// TIA Portal V19 export
DATA_BLOCK "InfeedPAC3200"   // DB19
TITLE = Instance DB of basic data collection
// Instance DB of basic data collection
// stored: InstanceOfName EnS_EnergyDataBasic, InstanceOfType FB
"EnS_EnergyDataBasic"
   // VAR_INPUT
   //    energyMeta : "EnS_typeEnergyMeta";
   //    energyBasic : "EnS_typeEnergyBasic";
   //    bufferDB { ExternalAccessible := 'False'; ExternalVisible := 'False'; ExternalWritable := 'False'} : DB_ANY;
   //    sD : Variant;
   //    messageSuppress { ExternalAccessible := 'False'; ExternalVisible := 'False'; ExternalWritable := 'False'} : Bool;
   // END_VAR
   // VAR_OUTPUT
   //    error { ExternalAccessible := 'False'; ExternalVisible := 'False'; ExternalWritable := 'False'} : Bool;
   //    errorAlarm1 { ExternalAccessible := 'False'; ExternalVisible := 'False'; ExternalWritable := 'False'} : Bool;
   //    errorAlarm2 { ExternalAccessible := 'False'; ExternalVisible := 'False'; ExternalWritable := 'False'} : Bool;
   //    errorAlarm3 { ExternalAccessible := 'False'; ExternalVisible := 'False'; ExternalWritable := 'False'} : Bool;
   //    alarmState1 { ExternalAccessible := 'False'; ExternalVisible := 'False'; ExternalWritable := 'False'} : Byte;
   //    alarmState2 { ExternalAccessible := 'False'; ExternalVisible := 'False'; ExternalWritable := 'False'} : Byte;
   //    alarmState3 { ExternalAccessible := 'False'; ExternalVisible := 'False'; ExternalWritable := 'False'} : Byte;
   //    status { ExternalAccessible := 'False'; ExternalVisible := 'False'; ExternalWritable := 'False'} : Word;
   //    status1 { ExternalAccessible := 'False'; ExternalVisible := 'False'; ExternalWritable := 'False'} : Word;
   //    status2 { ExternalAccessible := 'False'; ExternalVisible := 'False'; ExternalWritable := 'False'} : Word;
   //    status3 { ExternalAccessible := 'False'; ExternalVisible := 'False'; ExternalWritable := 'False'} : Word;
   //    statusAlarm1 { ExternalAccessible := 'False'; ExternalVisible := 'False'; ExternalWritable := 'False'} : Word;
   //    statusAlarm2 { ExternalAccessible := 'False'; ExternalVisible := 'False'; ExternalWritable := 'False'} : Word;
   //    statusAlarm3 { ExternalAccessible := 'False'; ExternalVisible := 'False'; ExternalWritable := 'False'} : Word;
   // END_VAR
   // VAR_IN_OUT
   //    orgData : "EnS_typeOrgData";
   //    bufferWork : "EnS_typeBufferWork";
   // END_VAR
   // VAR
   //    Program_Alarm1 { ExternalAccessible := 'False'; ExternalVisible := 'False'; ExternalWritable := 'False'; S7_SetPoint := 'True'} : Program_Alarm;
   //    Program_Alarm2 { ExternalAccessible := 'False'; ExternalVisible := 'False'; ExternalWritable := 'False'; S7_SetPoint := 'True'} : Program_Alarm;
   //    Program_Alarm3 { ExternalAccessible := 'False'; ExternalVisible := 'False'; ExternalWritable := 'False'; S7_SetPoint := 'True'} : Program_Alarm;
   //    ss_BufferWrite { ExternalAccessible := 'False'; ExternalVisible := 'False'; ExternalWritable := 'False'; S7_SetPoint := 'True'} : "EnS_BufferWrite";
   //    ss_DataEnergy { ExternalAccessible := 'False'; ExternalVisible := 'False'; ExternalWritable := 'False'; S7_SetPoint := 'True'} : "EnS_typeBufferWriteCtrl";
   //    ss_DataPower { ExternalAccessible := 'False'; ExternalVisible := 'False'; ExternalWritable := 'False'; S7_SetPoint := 'True'} : "EnS_typeBufferWriteCtrl";
   //    ss_DataEnergyCounter { ExternalAccessible := 'False'; ExternalVisible := 'False'; ExternalWritable := 'False'; S7_SetPoint := 'True'} : "EnS_typeBufferWriteCtrl";
   //    si16_CycleWrite { ExternalAccessible := 'False'; ExternalVisible := 'False'; ExternalWritable := 'False'} : Int;
   //    si16_CycleWriteAct { ExternalAccessible := 'False'; ExternalVisible := 'False'; ExternalWritable := 'False'} : Int;
   //    sbo_Write { ExternalAccessible := 'False'; ExternalVisible := 'False'; ExternalWritable := 'False'} : Bool;
   //    sbo_WriteEnergy { ExternalAccessible := 'False'; ExternalVisible := 'False'; ExternalWritable := 'False'} : Bool;
   //    sbo_WritePower { ExternalAccessible := 'False'; ExternalVisible := 'False'; ExternalWritable := 'False'} : Bool;
   //    sbo_WriteEnergyCounter { ExternalAccessible := 'False'; ExternalVisible := 'False'; ExternalWritable := 'False'} : Bool;
   //    sbo_WriteEnergyBusy { ExternalAccessible := 'False'; ExternalVisible := 'False'; ExternalWritable := 'False'} : Bool;
   //    sbo_WritePowerBusy { ExternalAccessible := 'False'; ExternalVisible := 'False'; ExternalWritable := 'False'} : Bool;
   //    sbo_WriteEnergyCounterBusy { ExternalAccessible := 'False'; ExternalVisible := 'False'; ExternalWritable := 'False'} : Bool;
   //    sbo_SyncPulseOld { ExternalAccessible := 'False'; ExternalVisible := 'False'; ExternalWritable := 'False'} : Bool;
   //    sbo_Alarm1 { ExternalAccessible := 'False'; ExternalVisible := 'False'; ExternalWritable := 'False'} : Bool;
   //    sbo_Alarm2 { ExternalAccessible := 'False'; ExternalVisible := 'False'; ExternalWritable := 'False'} : Bool;
   //    sbo_Alarm3 { ExternalAccessible := 'False'; ExternalVisible := 'False'; ExternalWritable := 'False'} : Bool;
   //    sbo_Alarm1Old { ExternalAccessible := 'False'; ExternalVisible := 'False'; ExternalWritable := 'False'} : Bool;
   //    sbo_Alarm2Old { ExternalAccessible := 'False'; ExternalVisible := 'False'; ExternalWritable := 'False'} : Bool;
   //    sbo_Alarm3Old { ExternalAccessible := 'False'; ExternalVisible := 'False'; ExternalWritable := 'False'} : Bool;
   //    sbo_ErrorAlarmState1 { ExternalAccessible := 'False'; ExternalVisible := 'False'; ExternalWritable := 'False'} : Bool;
   //    sbo_ErrorAlarmState2 { ExternalAccessible := 'False'; ExternalVisible := 'False'; ExternalWritable := 'False'} : Bool;
   //    sbo_ErrorAlarmState3 { ExternalAccessible := 'False'; ExternalVisible := 'False'; ExternalWritable := 'False'} : Bool;
   //    sbo_Init { ExternalAccessible := 'False'; ExternalVisible := 'False'; ExternalWritable := 'False'} : Bool;
   //    sb16_StatusAlarmState1 { ExternalAccessible := 'False'; ExternalVisible := 'False'; ExternalWritable := 'False'} : Word;
   //    sb16_StatusAlarmState2 { ExternalAccessible := 'False'; ExternalVisible := 'False'; ExternalWritable := 'False'} : Word;
   //    sb16_StatusAlarmState3 { ExternalAccessible := 'False'; ExternalVisible := 'False'; ExternalWritable := 'False'} : Word;
   // END_VAR
BEGIN
   energyMeta."name" := 'InfeedPAC3200';
   energyMeta.id[0] := 345;
   energyMeta.id[1] := 346;
   energyMeta.id[2] := 347;
   energyMeta.id[3] := 348;
   energyMeta.id[4] := 349;
   energyMeta.inputType := 2;
   energyMeta.configType := 2;
   energyMeta.mode := 1;
   energyMeta.syncPeriod := 60.0;
   energyMeta.overflowCntValue := 1000000.0;
   energyMeta.normFactorIn := 1.0;
   energyMeta.normFactorOut := 0.001;
   energyMeta.zeroCut := 0.0;
   energyMeta.baseAcqTime := 10.0;
   energyMeta.addAcqTime := 0.0;
   energyMeta.coordinationEnable := TRUE;
   energyMeta.cyclicRd := TRUE;
   energyMeta.cyclicTime := 10.0;
   energyMeta.unitActEnergy := 1179;
   energyMeta.unitActPower := 1190;
   energyMeta.unitAppEnergy := 1655;
   energyMeta.unitAppPower := 1652;
   energyMeta.unitReactEnergy := 1649;
   energyMeta.unitReactPower := 1646;
   energyMeta.unitPowerFactor := 1997;
   energyMeta.unitCurrent := 1209;
   energyMeta.unitVoltage := 1240;
   energyMeta.unitFrequency := 1077;
   energyMeta.unitAmpUnbalCurrent := 1342;
   energyMeta.unitAmpUnbalVoltage := 1342;
   energyMeta.archiveEnergy := TRUE;
   energyMeta.archivePower := TRUE;
   energyMeta.archiveEnergyCounter := TRUE;
END_DATA_BLOCK
